(* IEC 61131-3 sources: Word/plc-course/17-industrial-communications/labs/starter, 3 files *)

(* ---- 17-1-modbus-register-map.st ---- *)
(* Lab 17-1: Modbus register map for glycol skid GC-3.
   Module 17 (Industrial communications). STARTER - the declarations are done for you;
   write the logic where it says TODO, then run:
     python3 tools/plctest.py 17-industrial-communications/labs/starter/17-1-modbus-register-map.st

   You may add your own FUNCTIONs above the PROGRAM (for example one that joins two
   WORDs into a DINT). Keep every name in the interface table exactly as it is. *)

PROGRAM ModbusMap
  VAR (* field inputs *)
    PumpRunning AT %IX0.0 : BOOL;   (* P-301 running (contactor auxiliary contact) *)
    PumpFault   AT %IX0.1 : BOOL;   (* P-301 motor protection tripped *)
  END_VAR
  VAR (* holding registers served to SCADA. OpenPLC Runtime v3: %MW0 = holding register 1024 *)
    HR_Status   AT %MW0 : WORD;     (* PLC -> SCADA: status bits *)
    HR_Pressure AT %MW1 : INT;      (* PLC -> SCADA: PT-301 discharge pressure, bar x 100 *)
    HR_RunSecA  AT %MW2 : WORD;     (* PLC -> SCADA: RunSeconds, first register *)
    HR_RunSecB  AT %MW3 : WORD;     (* PLC -> SCADA: RunSeconds, second register *)
    HR_SupplySP AT %MW4 : INT := 50; (* SCADA -> PLC: glycol supply setpoint, degC x 10 *)
  END_VAR
  VAR (* registers read from flow meter FT-301 by the Modbus client *)
    MeterRegA AT %IW100 : WORD;     (* first register of the meter's totaliser *)
    MeterRegB AT %IW101 : WORD;     (* second register of the meter's totaliser *)
  END_VAR
  VAR (* the PLC side of the map *)
    PressureBar     : REAL;         (* PT-301 pressure in bar, from the analog input scaling *)
    RunSeconds      : DINT;         (* P-301 running time in seconds *)
    RunSecLowFirst  : BOOL;         (* FALSE: HR_RunSecA = high word. TRUE: HR_RunSecA = low word *)
    MeterLowFirst   : BOOL;         (* same meaning for MeterRegA / MeterRegB *)
    MeterTotal      : DINT;         (* FT-301 totaliser in litres *)
    SupplySP        : REAL := 5.0;  (* glycol supply setpoint in use, degC *)
    PressOutOfRange : BOOL;         (* pressure did not fit in HR_Pressure and was clamped *)
    SPRejected      : BOOL;         (* HR_SupplySP holds a value outside -10.0 .. +15.0 degC *)
  END_VAR

  (* TODO 1: split RunSeconds into HR_RunSecA / HR_RunSecB (word order: RunSecLowFirst).
     TODO 2: join MeterRegA / MeterRegB into MeterTotal (word order: MeterLowFirst).
     TODO 3: PressureBar -> HR_Pressure (x 100, rounded), clamp and set PressOutOfRange.
     TODO 4: HR_SupplySP -> SupplySP (/ 10) if -100..150, otherwise keep it and set SPRejected.
     TODO 5: build HR_Status from PumpRunning, PumpFault, PressOutOfRange, SPRejected.
     Replace these placeholder lines with your logic. *)
  HR_Status := 16#0000;
  HR_Pressure := 0;
  MeterTotal := 0;
END_PROGRAM

CONFIGURATION Config0
  RESOURCE Res0 ON PLC
    TASK MainTask(INTERVAL := T#10ms, PRIORITY := 0);
    PROGRAM Inst0 WITH MainTask : ModbusMap;
  END_RESOURCE
END_CONFIGURATION

(* ---- 17-2-comm-watchdog.st ---- *)
(* Lab 17-2: Communication watchdog for a reservoir telemetry link.
   Module 17 (Industrial communications). STARTER - the declarations are done for you;
   write the logic where it says TODO, then run:
     python3 tools/plctest.py 17-industrial-communications/labs/starter/17-2-comm-watchdog.st

   Pump station PS-1 fills reservoir R-2 over a radio link. The Modbus client polls the
   reservoir outstation about once a second and leaves the last values it received in
   %IW100..%IW102, so if the link fails those values simply FREEZE.

   This is a training exercise, not a design for a real overfill protection. *)

PROGRAM CommWatchdog
  VAR (* data from the reservoir outstation, placed here by the Modbus client *)
    RxHeartbeat AT %IW100 : INT;    (* outstation heartbeat: +1 every second *)
    RxLevel     AT %IW101 : INT;    (* reservoir level, % x 10 (0..1000) *)
    RxStatus    AT %IW102 : WORD;   (* bit 0: reservoir inlet valve open *)
  END_VAR
  VAR (* data to the outstation *)
    TxHeartbeat AT %QW100 : INT;    (* our heartbeat: +1 every second *)
  END_VAR
  VAR (* field output *)
    FillPump AT %QX0.0 : BOOL;      (* fill pump P-1 run command *)
  END_VAR
  VAR (* results *)
    CommLost  : BOOL := TRUE;       (* TRUE: the received data cannot be trusted *)
    LossCount : INT;                (* number of healthy -> lost transitions *)
    LevelPct  : REAL := 100.0;      (* level used by the control logic, % *)
    InletOpen : BOOL;               (* inlet valve state used by the control logic *)
  END_VAR
  VAR
    (* TODO: add the timers and other internal variables you need here. *)
    LastBeat : INT;                 (* heartbeat value seen on the previous scan *)
  END_VAR

  (* TODO 1: our own heartbeat: TxHeartbeat + 1 every second; after 32767 it goes to 0.
     TODO 2: supervise RxHeartbeat: CommLost TRUE 3 s after the last change; FALSE again
             only after the heartbeat has kept changing for 5 s. Count each loss once.
     TODO 3: LevelPct / InletOpen: live values, or the fallback values while CommLost.
     TODO 4: FillPump: start below 40 %, stop at 90 %, stop if CommLost or inlet closed.
     Replace these placeholder lines with your logic. *)
  LastBeat := RxHeartbeat;
  FillPump := FALSE;
END_PROGRAM

CONFIGURATION Config0
  RESOURCE Res0 ON PLC
    TASK MainTask(INTERVAL := T#10ms, PRIORITY := 0);
    PROGRAM Inst0 WITH MainTask : CommWatchdog;
  END_RESOURCE
END_CONFIGURATION

(* ---- 17-3-drive-control-word.st ---- *)
(* Lab 17-3: Drive control word and status word (simplified generic drive profile).
   Module 17 (Industrial communications). STARTER - the declarations are done for you;
   write the logic where it says TODO, then run:
     python3 tools/plctest.py 17-industrial-communications/labs/starter/17-3-drive-control-word.st

   The bit layout is the course's SIMPLIFIED GENERIC PROFILE (see the lesson), not
   PROFIdrive, CiA 402 or the ODVA profile.

   Control word (PLC -> drive)          Status word (drive -> PLC)
     bit 0  RUN    1 = run, 0 = stop       bit 0  READY     healthy, will run on RUN
     bit 1  REV    1 = reverse             bit 1  RUNNING   output active
     bit 2  RESET  acts on 0 -> 1          bit 2  FAULT     tripped
     bits 3-15     always 0                bit 3  AT_SPEED  actual = reference
                                           bits 4-15        vendor-specific, ignored
   Speed reference: 0..16384 = 0..100 % of maximum speed. *)

PROGRAM DriveProfile
  VAR (* field input *)
    ResetPB AT %IX0.0 : BOOL;       (* fault reset push-button, NO *)
  END_VAR
  VAR (* fieldbus input data from the drive *)
    DriveSts AT %IW100 : WORD;      (* status word *)
  END_VAR
  VAR (* fieldbus output data to the drive *)
    DriveCtrl     AT %QW100 : WORD; (* control word *)
    DriveSpeedRef AT %QW101 : INT;  (* speed reference, 16384 = 100 % *)
  END_VAR
  VAR (* requests from the conveyor sequence *)
    RunReq  : BOOL;                 (* TRUE = the drive should run *)
    RevReq  : BOOL;                 (* TRUE = reverse direction wanted *)
    SpeedSP : REAL;                 (* speed setpoint, % of maximum *)
  END_VAR
  VAR (* decoded status for the sequence and the HMI *)
    Ready     : BOOL;
    Running   : BOOL;
    Faulted   : BOOL;
    AtSpeed   : BOOL;
    StartFail : BOOL;               (* latched: RUN sent but no RUNNING within 3 s *)
  END_VAR
  VAR
    (* TODO: add the edge detector, timers and internal flags you need here. *)
    Ctrl : WORD;                    (* control word under construction *)
  END_VAR

  (* TODO 1: decode Ready / Running / Faulted / AtSpeed from DriveSts.
     TODO 2: fault reset: one 500 ms RESET pulse per press; the press also clears StartFail.
     TODO 3: StartFail: RUN sent for 3 s without RUNNING.
     TODO 4: RUN bit from RunReq, blocked by a fault or StartFail; a request that saw a
             fault is spent until RunReq has been released.
     TODO 5: REV bit from RevReq, only while the drive is not RUNNING.
     TODO 6: build DriveCtrl; bits 3..15 always 0.
     TODO 7: DriveSpeedRef from SpeedSP (clamp 0..100 %, 100 % = 16384).
     Replace these placeholder lines with your logic. *)
  Ctrl := 16#0000;
  DriveCtrl := Ctrl;
  DriveSpeedRef := 0;
END_PROGRAM

CONFIGURATION Config0
  RESOURCE Res0 ON PLC
    TASK MainTask(INTERVAL := T#10ms, PRIORITY := 0);
    PROGRAM Inst0 WITH MainTask : DriveProfile;
  END_RESOURCE
END_CONFIGURATION
